FUNCTION F_TargetReachedOrHigher : BOOL
VAR_INPUT
	fCurrentPos: LREAL;
	fTargetPos: LREAL;
END_VAR


F_TargetReachedOrHigher := fCurrentPos >= (fTargetPos - fEpsilon);

END_FUNCTION

(* stored: Version 1.1.0.1, ProductVersion 3.1.4020.12
   POU F_TargetReachedOrHigher: Id {00ddc253-e675-4b1f-98a1-5439eb7a1734}, SpecialFunc None *)
